PROGRAM MAIN
VAR    
    {attribute 'pytmc' := '
        pv: RM113
    '}
    {attribute 'TcLinkTo' := '.iRaw := TIIB[Term 3 (EL3202-0010)]^RTD Inputs Channel 1^Value'}
    fbTempSensor : FB_TempSensor;
    fTemp : LREAL;
    
    {attribute 'pytmc' := '
        pv: RM113
    '}
    fbFlutterDet : FB_FlutterDetection;
    bTestFlip : BOOL;

    fbTrigTest : FB_TestTrigger;
    
END_VAR

fbTempSensor(fResolution:=0.01);

fTemp := fbTempSensor.fTemp;
fTemp := (9.0/5.0) * fTemp + 32;

fbFlutterDet(fPastTime:=T#5000ms, bVarToMonitor:=bTestFlip);
//fbTrigTest(bTestBool:=bTestFlip);

END_PROGRAM

(* stored: Version 1.1.0.1, ProductVersion 3.1.4022.18
   POU MAIN: Id {2fb27e99-f448-43cc-be37-ad260877f38c}, SpecialFunc None *)
